// TIA Portal V20 export
DATA_BLOCK "BK08"   // DB234
// stored: MemoryReserve 100
   VAR
      "X10-1 TOP TAPE CLAMP TOP LEFT UP" : Bool;
      "X11-1 TOP TAPE CLAMP TOP CENTER UP" : Bool;
      "X12-1 TOP TAPE CLAMP TOP RIGHT UP" : Bool;
      "X13-1 TOP TAPE ATTACHMENT VACUUM PRESSURE SWITCH" : Bool;
      "X14-1 TOP TAPE CLAMP BTM DOWN" : Bool;
      "X15-1 TOP TAPING Y-AXIS LIMIT SENSOR(-)" : Bool;
      "X16-1 TOP TAPING Y-AXIS LIMIT SENSOR(+)" : Bool;
      "X17-1 TOP TAPE FIX STAGE STACK DETECT SENSOR" : Bool;
      "X10-2 TOP TAPE CLAMP TOP LEFT DOWN" : Bool;
      "X11-2 TOP TAPE CLAMP TOP CENTER DOWN" : Bool;
      "X12-2 TOP TAPE CLAMP TOP RIGHT DOWN" : Bool;
      "X13-2 SPARE" : Bool;
      "X14-2 TOP TAPE CLAMP BTM UP" : Bool;
      "X15-2 TOP TAPING Y-AXIS HOME SENSOR" : Bool;
      "X16-2 SPARE" : Bool;
      "X17-2 SPARE" : Bool;
   END_VAR
BEGIN
END_DATA_BLOCK
